{attribute 'enable_dynamic_creation'}
{attribute 'no_explicit_call' := 'do not call this FB directly'}
FUNCTION_BLOCK PUBLIC FileEntry EXTENDS FileSystemEntry IMPLEMENTS I_FileEntry
VAR	
	_name : FileName;
END_VAR

METHOD FB_init : BOOL
VAR_INPUT
	bInitRetains : BOOL; // if TRUE, the retain variables are initialized (warm start / cold start)
	bInCopyCode : BOOL;  // if TRUE, the instance afterwards gets moved into the copy code (online change)
	Path : FilePath;
	Name : FileName;
END_VAR
SUPER^.FB_init(bInitRetains,bInCopyCode,Path);
THIS^._name := Name;
END_METHOD

METHOD GetFullPath : T_MaxString
VAR
	fullPath : T_MaxString;
END_VAR
fullPath := CONCAT(fullPath, Path);
fullPath := CONCAT(fullPath, Name);

GetFullPath := fullPath;
END_METHOD

PROPERTY PUBLIC IsFile : BOOL
GET
IsFile := TRUE;
END_GET
END_PROPERTY

PROPERTY Name : FileName
GET
Name := _name;
END_GET
SET
_name := Name;
END_SET
END_PROPERTY

END_FUNCTION_BLOCK

(* stored: Version 1.1.0.1, ProductVersion 3.1.4024.9
   POU FileEntry: Id {2d354d0c-5b37-4387-b88a-8916d5810531}, SpecialFunc None
   Folder Constructor: Id {ae4d46b4-5374-4aa2-831e-ccf5bdf63bf8}
   Method FB_init: Id {5bb46322-f6e4-4e47-ae98-4856388d9411}
   Method GetFullPath: Id {86dfb3ba-2ac4-453b-9589-99870abc7f47}
   Property IsFile: Id {33e44ebc-1a90-4c27-b7ae-5c4ddac8c9bf}
   Get Get: Id {ae20e2e8-62bb-4a05-903f-7804483bda5f}
   Property Name: Id {98db7d2a-7a90-4828-a6fa-6391ab557d8f}
   Get Get: Id {306ee5b5-bc75-4317-b5d1-9a0654270ce7}
   Set Set: Id {add0cd59-73db-4c0d-8b1d-42544f91ba8c} *)
